{attribute 'GeneratedUsingTerminal: EL3311-0000-0018'}
{attribute addProperty BoxType "EL3311-0000-0018"}
{attribute addProperty Id "TC_InputsAT %I*TC_Inputs_4A3944819WcStateAT %I*WcState_9091E0EB2InfoDataAT %I*InfoData_94A18F5E2"}
{attribute addProperty CRC "2665756135"}
{attribute addProperty Size "13"}
TYPE EL3311_9EE435E7 EXTENDS EtcSlaveTerminalBase_947E5A46 :
STRUCT
	{attribute addProperty Name "TC_Inputs"}
	TC_Inputs : TC_Inputs_4A394481;
	{attribute addProperty Name "WcState"}
	WcState : WcState_9091E0EB;
	{attribute addProperty Name "InfoData"}
	InfoData : InfoData_94A18F5E;
END_STRUCT
END_TYPE

(* stored: Version 1.2.0.0, ProductVersion 3.1.4024.9
   DUT EL3311_9EE435E7: Id {a5bd0673-c9b1-40bc-a52d-eb755bdda80c} *)
